{attribute 'linkalways'} 
{attribute 'no_explicit_call' := 'This FB is a CLASS and must be accessed using methods or properties'}
{attribute 'enable_dynamic_creation'}
FUNCTION_BLOCK _TcVnRectangle_DINT EXTENDS StructuredDatatypeBase
VAR
	localData : TcVnRectangle_DINT;
	activeData : REFERENCE TO TcVnRectangle_DINT REF= localData;
	_nX : _DINT(localData.nX);
	_nY : _DINT(localData.nY);
    _nWidth : _DINT(localData.nWidth);
	_nHeight : _DINT(localData.nHeight);
END_VAR

PROPERTY PUBLIC Address : PVOID
GET
Address := ADR(activeData);
END_GET
END_PROPERTY

METHOD PUBLIC ClearReference
VAR_INPUT
END_VAR
activeData REF= localData;
SetMemberReference();
END_METHOD

METHOD PUBLIC Clone : I_Datatype
VAR
    pClone : POINTER TO _TcVnRectangle_DINT;
END_VAR
pClone := __NEW(_TcVnRectangle_DINT());
pClone^.Value := Value;
Clone := pClone^;
END_METHOD

METHOD FB_init : BOOL
VAR_INPUT
	bInitRetains : BOOL; // if TRUE, the retain variables are initialized (warm start / cold start)
	bInCopyCode : BOOL;  // if TRUE, the instance afterwards gets moved into the copy code (online change)
END_VAR
SetMemberReference();
AddMember('nX',_nX);
AddMember('nY',_nY);
AddMember('nWidth',_nWidth);
AddMember('nHeight',_nHeight);
END_METHOD

PROPERTY PUBLIC Identifier : T_MAXSTRING
GET
Identifier := 'TcVnRectangle_DINT';
END_GET
END_PROPERTY

METHOD PUBLIC MakeReferenceTo
VAR_INPUT
	ReferenceTarget : REFERENCE TO TcVnRectangle_DINT;
END_VAR
activeData REF= ReferenceTarget;
SetMemberReference();
END_METHOD

PROPERTY PUBLIC nHeight : REFERENCE TO _DINT
GET
nHeight REF= _nHeight;
END_GET
END_PROPERTY

PROPERTY PUBLIC nWidth : REFERENCE TO _DINT
GET
nWidth REF= _nWidth;
END_GET
END_PROPERTY

PROPERTY PUBLIC nX : REFERENCE TO _DINT
GET
nX REF= _nX;
END_GET
END_PROPERTY

PROPERTY PUBLIC nY : REFERENCE TO _DINT
GET
nY REF= _nY;
END_GET
END_PROPERTY

METHOD PROTECTED SetMemberReference
VAR_INPUT
END_VAR
_nX.MakeReferenceTo(activeData.nX);
_nY.MakeReferenceTo(activeData.nY);
_nWidth.MakeReferenceTo(activeData.nWidth);
_nHeight.MakeReferenceTo(activeData.nHeight);
END_METHOD

PROPERTY PUBLIC Size : UDINT
GET
Size := SIZEOF(activeData);
END_GET
END_PROPERTY

METHOD TryMakeReferenceTo : BOOL
VAR_INPUT
	Target : I_Datatype;
END_VAR
VAR
	targetAsStruct : I_StructuredDatatype;
	pTargetData : POINTER TO TcVnRectangle_DINT;
END_VAR
IF NOT Target.TryResolveAsStructuredDatatype(targetAsStruct) THEN
	RETURN;
END_IF

IF NOT (targetAsStruct.Identifier = Identifier) THEN
	RETURN;
END_IF

pTargetData := Target.Address;
activeData REF= pTargetData^;
SetMemberReference();
TryMakeReferenceTo := TRUE;
END_METHOD

PROPERTY PUBLIC Value : REFERENCE TO TcVnRectangle_DINT
GET
Value REF= activeData;
END_GET
END_PROPERTY

END_FUNCTION_BLOCK

(* stored: Version 1.1.0.1, ProductVersion 3.1.4024.13
   POU _TcVnRectangle_DINT: Id {3ca0b904-c59f-0e94-3333-d42f0831b594}, SpecialFunc None
   Folder Constructor: Id {95e10b9e-86a5-0970-3d8f-27b2b3b12c0d}
   Folder Protected: Id {edd2a2dc-5a0c-0697-13a3-e302a13daa19}
   Property Address: Id {58d38feb-44a5-07f0-26aa-15ea57315367}
   Get Get: Id {d8777cb8-e1fd-07a5-389c-9d4db206f201}
   Method ClearReference: Id {24a48758-8b7d-0165-3c4c-c9a286d657d6}
   Method Clone: Id {348f7a38-f503-0292-21c1-c93dba95eb8a}
   Method FB_init: Id {e0ba2884-9f47-0df5-188d-ca70bc9d4ae8}
   Property Identifier: Id {4984899f-e331-0f86-2b66-e5347065a358}
   Get Get: Id {766c954a-6002-0c48-37bf-373dd989d68e}
   Method MakeReferenceTo: Id {290d5b35-2e28-0755-1c88-b8fa5e076da5}
   Property nHeight: Id {cdc73b3f-36a0-0319-3782-1fdcfa145e5f}
   Get Get: Id {1f82ce09-8032-02f7-020f-2c9c5cd13be4}
   Property nWidth: Id {8601aa17-6ebc-0132-3308-4b93d0acb078}
   Get Get: Id {8330d8ae-a546-0cbe-08a5-24b5aed9610e}
   Property nX: Id {6ea5cba2-6b3e-06e5-2d8c-fdbef3d02940}
   Get Get: Id {f89e643b-4f6b-06fd-372e-d8de1dea8280}
   Property nY: Id {2b7fdd00-13bf-0fec-2323-86e1c6d802c0}
   Get Get: Id {85171e6e-adfb-0bc2-39b8-2a374f53c330}
   Method SetMemberReference: Id {5c99d35d-0153-0b0a-14d6-cb7cc2a42480}
   Property Size: Id {bc97b1c1-00f1-074e-01a5-88c95d018dfa}
   Get Get: Id {960ec335-8590-0529-0678-3afee61124da}
   Method TryMakeReferenceTo: Id {26eecf6e-dff7-0609-1ee5-d42bc3e6aa2c}
   Property Value: Id {3c49b5ed-d289-03a1-2016-5083665b03d0}
   Get Get: Id {8bd9156a-7689-07f1-0c0a-3b991fe5fbba} *)
